(* CODESYS project main.project

Project tree, tasks and I/O mapping:
  Device : CODESYS Control Win V3, 3S - Smart Software Solutions GmbH, order no. 305021, version 3.5.8.30
    application Application
      libraries: Standard, * (System)
      task MainTask (cyclic, interval t#20ms, priority 1) calls PLC_PRG
      program PLC_PRG [ST]
    Modbus_COM : Modbus COM, 3S - Smart Software Solutions GmbH, version 3.4.0.0
        settings: DataBits = 8; StopBits = 2; ComPort = 3
      Modbus_Master_COM_Port : Modbus Master, COM Port, 3S - Smart Software Solutions GmbH, version 3.5.8.10
          settings: Transmission = 'RTU'; ResponseTimeout = 10; TimeBetweenFrames = 0; Auto-restart communication = TRUE
        Modbus_Slave_COM_Port : Modbus Slave, COM Port, 3S - Smart Software Solutions GmbH, version 3.5.4.0
            settings: SlaveAddress = 10; ResponseTimeout = 2; UseExtendedFunctionCodes = TRUE; Channel 0.Function Code = 2; Channel 0.Read Offset = 16#0000; Channel 0.Read Length = 32; Channel 0.Write Offset = 0; Channel 0.Write Length = 0; Channel 0.Cycle Time = 5; Channel 1.Function Code = 15; Channel 1.Read Offset = 0; Channel 1.Read Length = 0; Channel 1.Write Offset = 16#0000; Channel 1.Write Length = 32; Channel 1.Cycle Time = 5; Channel 2.Function Code = 6; Channel 2.Read Offset = 0; Channel 2.Read Length = 0; Channel 2.Write Offset = 16#0012; Channel 2.Write Length = 1; Channel 2.Cycle Time = 100
            input  I0 : BOOL  // Channel 0.Channel 0.Bit0
            input  I13 : BOOL  // Channel 0.Channel 0.Bit5
            input  I14 : BOOL  // Channel 0.Channel 0.Bit6
            input  I15 : BOOL  // Channel 0.Channel 0.Bit7
            input  out0Vcc : BOOL  // Channel 0.Channel 0.Bit4
            input  out1Vcc : BOOL  // Channel 0.Channel 0.Bit5
            input  out0DiagRaw : BOOL  // Channel 0.Channel 0.Bit6
            input  out1DiagRaw : BOOL  // Channel 0.Channel 0.Bit7
            input  inRunSwitch : BOOL  // Channel 0.Channel 0.Bit0
            input  isRun : BOOL  // Channel 0.Channel 0.Bit1
            input  out0ErrorFlag : BOOL  // Channel 0.Channel 0.Bit2
            input  out1ErrorFlag : BOOL  // Channel 0.Channel 0.Bit3
            input  timeoutErrorFlag : BOOL  // Channel 0.Channel 0.Bit4
            output Y0 : BOOL  // Channel 1.Channel 1.Bit0
            output Y1 : BOOL  // Channel 1.Channel 1.Bit1
            output Y2 : BOOL  // Channel 1.Channel 1.Bit2
            output Y3 : BOOL  // Channel 1.Channel 1.Bit3
            output Y4 : BOOL  // Channel 1.Channel 1.Bit4
            output Y5 : BOOL  // Channel 1.Channel 1.Bit5
            output Y6 : BOOL  // Channel 1.Channel 1.Bit6
            output Y7 : BOOL  // Channel 1.Channel 1.Bit7
            output Y8 : BOOL  // Channel 1.Channel 1.Bit0
            output Y9 : BOOL  // Channel 1.Channel 1.Bit1
            output Y10 : BOOL  // Channel 1.Channel 1.Bit2
            output Y11 : BOOL  // Channel 1.Channel 1.Bit3
            output Y12 : BOOL  // Channel 1.Channel 1.Bit4
            output Y13 : BOOL  // Channel 1.Channel 1.Bit5
            output Y14 : BOOL  // Channel 1.Channel 1.Bit6
            output Y15 : BOOL  // Channel 1.Channel 1.Bit7
            output Run : BOOL  // Channel 1.Channel 1.Bit0
            output ResetError : BOOL  // Channel 1.Channel 1.Bit1
            output saveOutInStop : BOOL  // Channel 1.Channel 1.Bit2
            output timeoutCounter : WORD  // Channel 2.Channel 2
            unmapped channels: Channel 0, Channel 1, Channel 2
        Modbus_Slave_COM_Port_1 : Modbus Slave, COM Port, 3S - Smart Software Solutions GmbH, version 3.5.4.0
            settings: SlaveAddress = 11; ResponseTimeout = 100; UseExtendedFunctionCodes = TRUE; Channel 0.Function Code = 15; Channel 0.Read Offset = 0; Channel 0.Read Length = 0; Channel 0.Write Offset = 16#0000; Channel 0.Write Length = 12; Channel 0.Cycle Time = 5; Channel 1.Function Code = 6; Channel 1.Read Offset = 0; Channel 1.Read Length = 0; Channel 1.Write Offset = 16#000F; Channel 1.Write Length = 1; Channel 1.Cycle Time = 100
            output test11 : BYTE  // Channel 0.Channel 0
            output Q111 : BOOL  // Channel 0.Channel 0.Bit3
            output run11 : WORD  // Channel 1.Channel 1
            unmapped channels: Channel 0, Channel 1
*)

// Device/Application/PLC_PRG
PROGRAM PLC_PRG
VAR
	counter : INT := 0;
	rTrigI0 : R_TRIG;
	fTrigI0 : F_TRIG;
	rTrigModbusError : R_TRIG;
END_VAR

rTrigModbusError( clk := Modbus_Slave_COM_Port.xError );
Modbus_Slave_COM_Port( xReset := rTrigModbusError.Q );

rTrigI0( clk := I0 );
fTrigI0( clk := I0 );

// Set Modbus timeout:
timeoutCounter := 500;

// Auto clear output bits in stop ( but if not Run then out is in 0 )
// ( Само за тестване дали се адресират правилните изходи без физически изход )  
saveOutInStop := FALSE;

IF I14 AND ( out1ErrorFlag OR out0ErrorFlag OR timeoutErrorFlag ) THEN
	IF ( out0DiagRaw AND out0Vcc ) AND ( out1DiagRaw AND out1Vcc) THEN
		ResetError := 1;
	END_IF
ELSE
		ResetError := 0;
END_IF

IF I15 = TRUE THEN
	Run := FALSE;
END_IF

IF I14 AND isRun = FALSE THEN
	IF ( out0Vcc AND out0DiagRaw ) AND ( out1Vcc AND out1DiagRaw ) THEN 
		Run := TRUE;
		counter := 0;
	END_IF
END_IF

IF rTrigI0.Q or fTrigI0.Q THEN
	counter := counter + 1;
	IF counter > 255 THEN
		counter := 0;
	END_IF
END_IF

Y1 := NOT( I0 );
Y2 := I0;

Y8 := counter.0;
Y9 := counter.1;
Y10 := counter.2;
Y11 := counter.3;
Y12 := counter.4;
Y13 := counter.5;
Y14 := counter.6;
Y15 := counter.7;

run11.0 := Run;
Q111 := I13;
test11.0 := counter.0;
test11.1 := counter.1;
test11.2 := counter.2;
test11.3 := counter.3;
test11.4 := counter.4;
test11.5 := counter.5;
test11.6 := counter.6;
test11.7 := counter.7;

END_PROGRAM
